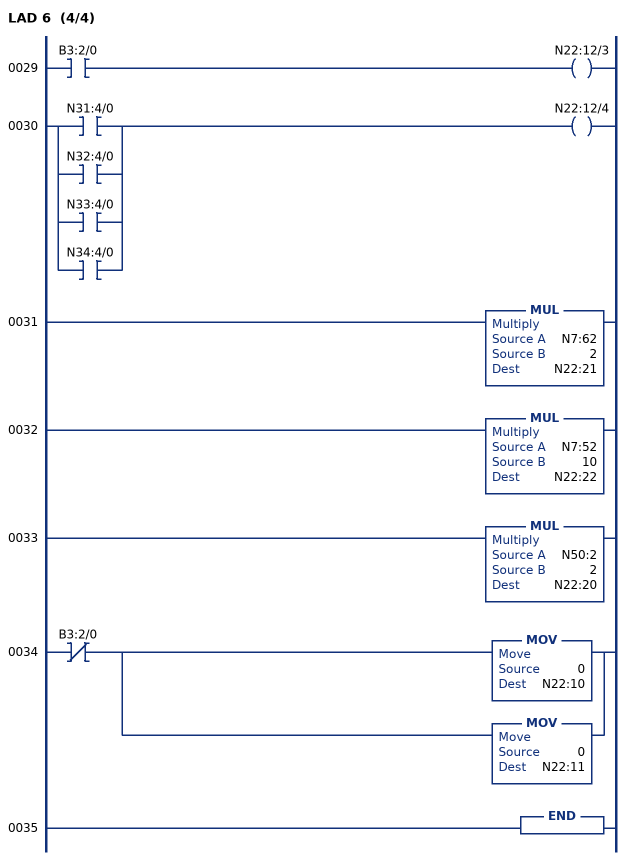
% Rung: 29 %
SOR XIC B3:2/0 OTE N22:12/3 EOR
% Rung: 30 %
SOR BST XIC N31:4/0 NXB XIC N32:4/0 NXB XIC N33:4/0 NXB XIC N34:4/0 BND OTE N22:12/4 EOR
% Rung: 31 %
SOR MUL N7:62 2 N22:21 EOR
% Rung: 32 %
SOR MUL N7:52 10 N22:22 EOR
% Rung: 33 %
SOR MUL N50:2 2 N22:20 EOR
% Rung: 34 %
SOR XIO B3:2/0 BST MOV 0 N22:10 NXB MOV 0 N22:11 BND EOR
% Rung: 35 %
SOR END EOR

LADDER 7
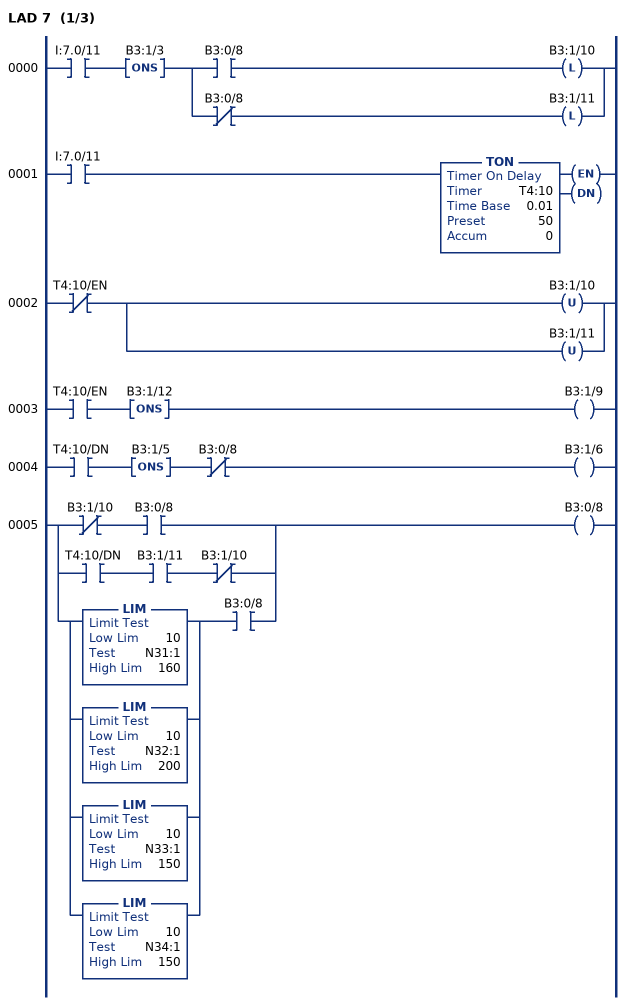
% Rung: 0 %
SOR XIC I:7.0/11 OSR B3:1/3 BST XIC B3:0/8 OTL B3:1/10 NXB XIO B3:0/8 OTL B3:1/11 BND EOR
% Rung: 1 %
SOR XIC I:7.0/11 TON T4:10 0.01 50 0 EOR
% Rung: 2 %
SOR XIO T4:10/EN BST OTU B3:1/10 NXB OTU B3:1/11 BND EOR
% Rung: 3 %
SOR XIC T4:10/EN OSR B3:1/12 OTE B3:1/9 EOR
% Rung: 4 %
SOR XIC T4:10/DN OSR B3:1/5 XIO B3:0/8 OTE B3:1/6 EOR
% Rung: 5 %
SOR BST BST XIO B3:1/10 XIC B3:0/8 NXB XIC T4:10/DN XIC B3:1/11 XIO B3:1/10 BND NXB BST LIM 10 N31:1 160 NXB LIM 10 N32:1 200 NXB LIM 10 N33:1 150 NXB LIM 10 N34:1 150 BND XIC B3:0/8 BND OTE B3:0/8 EOR

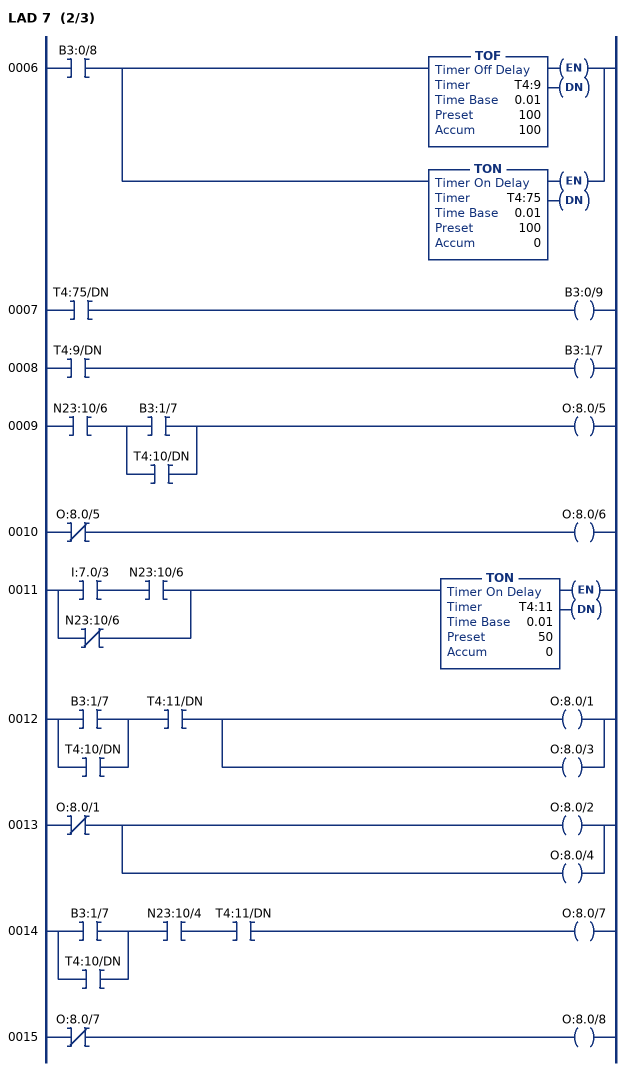
% Rung: 6 %
SOR XIC B3:0/8 BST TOF T4:9 0.01 100 100 NXB TON T4:75 0.01 100 0 BND EOR
% Rung: 7 %
SOR XIC T4:75/DN OTE B3:0/9 EOR
% Rung: 8 %
SOR XIC T4:9/DN OTE B3:1/7 EOR
% Rung: 9 %
SOR XIC N23:10/6 BST XIC B3:1/7 NXB XIC T4:10/DN BND OTE O:8.0/5 EOR
% Rung: 10 %
SOR XIO O:8.0/5 OTE O:8.0/6 EOR
% Rung: 11 %
SOR BST XIC I:7.0/3 XIC N23:10/6 NXB XIO N23:10/6 BND TON T4:11 0.01 50 0 EOR
% Rung: 12 %
SOR BST XIC B3:1/7 NXB XIC T4:10/DN BND XIC T4:11/DN BST OTE O:8.0/1 NXB OTE O:8.0/3 BND EOR
% Rung: 13 %
SOR XIO O:8.0/1 BST OTE O:8.0/2 NXB OTE O:8.0/4 BND EOR
% Rung: 14 %
SOR BST XIC B3:1/7 NXB XIC T4:10/DN BND XIC N23:10/4 XIC T4:11/DN OTE O:8.0/7 EOR
% Rung: 15 %
SOR XIO O:8.0/7 OTE O:8.0/8 EOR

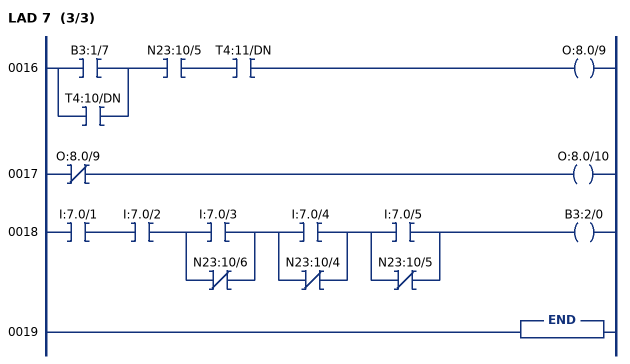
% Rung: 16 %
SOR BST XIC B3:1/7 NXB XIC T4:10/DN BND XIC N23:10/5 XIC T4:11/DN OTE O:8.0/9 EOR
% Rung: 17 %
SOR XIO O:8.0/9 OTE O:8.0/10 EOR
% Rung: 18 %
SOR XIC I:7.0/1 XIC I:7.0/2 BST XIC I:7.0/3 NXB XIO N23:10/6 BND BST XIC I:7.0/4 NXB XIO N23:10/4 BND BST XIC I:7.0/5 NXB XIO N23:10/5 BND OTE B3:2/0 EOR
% Rung: 19 %
SOR END EOR

LADDER 8
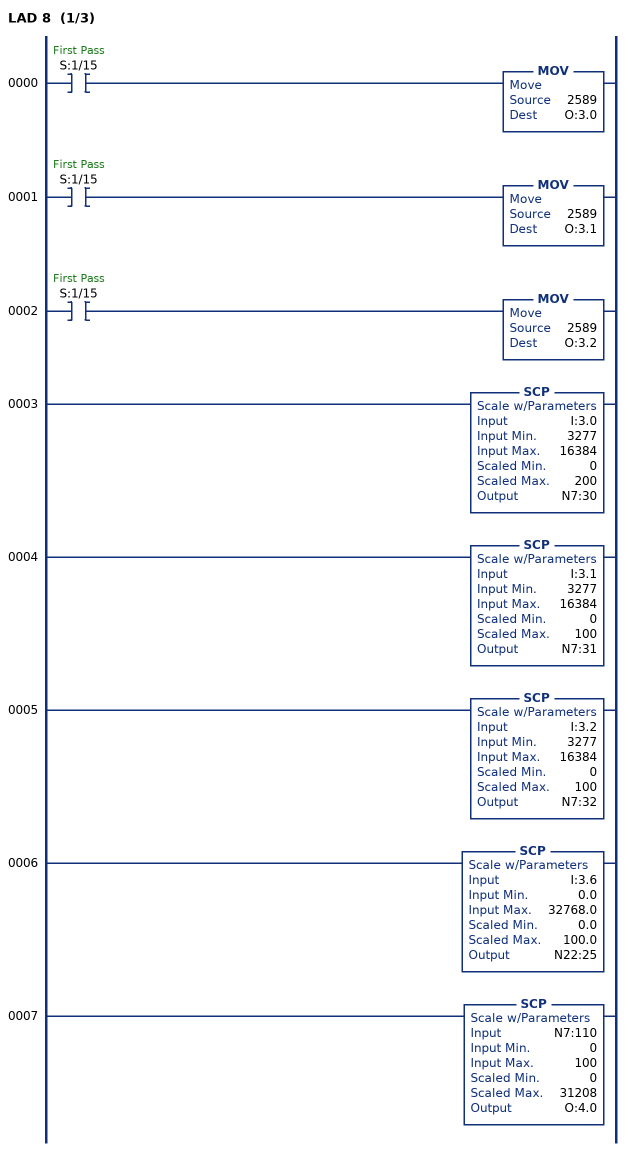
% Rung: 0 %
SOR XIC S:1/15 MOV 2589 O:3.0 EOR
%   S:1/15  "First Pass" %
% Rung: 1 %
SOR XIC S:1/15 MOV 2589 O:3.1 EOR
%   S:1/15  "First Pass" %
% Rung: 2 %
SOR XIC S:1/15 MOV 2589 O:3.2 EOR
%   S:1/15  "First Pass" %
% Rung: 3 %
SOR SCP I:3.0 3277 16384 0 200 N7:30 EOR
% Rung: 4 %
SOR SCP I:3.1 3277 16384 0 100 N7:31 EOR
% Rung: 5 %
SOR SCP I:3.2 3277 16384 0 100 N7:32 EOR
% Rung: 6 %
SOR SCP I:3.6 0.0 32768.0 0.0 100.0 N22:25 EOR
% Rung: 7 %
SOR SCP N7:110 0 100 0 31208 O:4.0 EOR

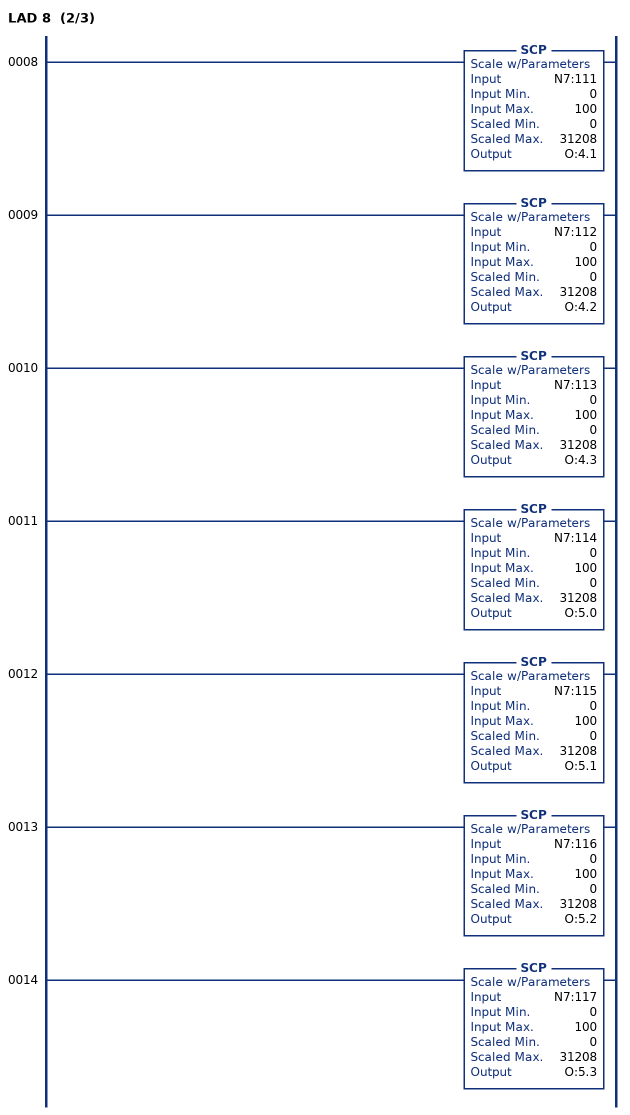
% Rung: 8 %
SOR SCP N7:111 0 100 0 31208 O:4.1 EOR
% Rung: 9 %
SOR SCP N7:112 0 100 0 31208 O:4.2 EOR
% Rung: 10 %
SOR SCP N7:113 0 100 0 31208 O:4.3 EOR
% Rung: 11 %
SOR SCP N7:114 0 100 0 31208 O:5.0 EOR
% Rung: 12 %
SOR SCP N7:115 0 100 0 31208 O:5.1 EOR
% Rung: 13 %
SOR SCP N7:116 0 100 0 31208 O:5.2 EOR
% Rung: 14 %
SOR SCP N7:117 0 100 0 31208 O:5.3 EOR

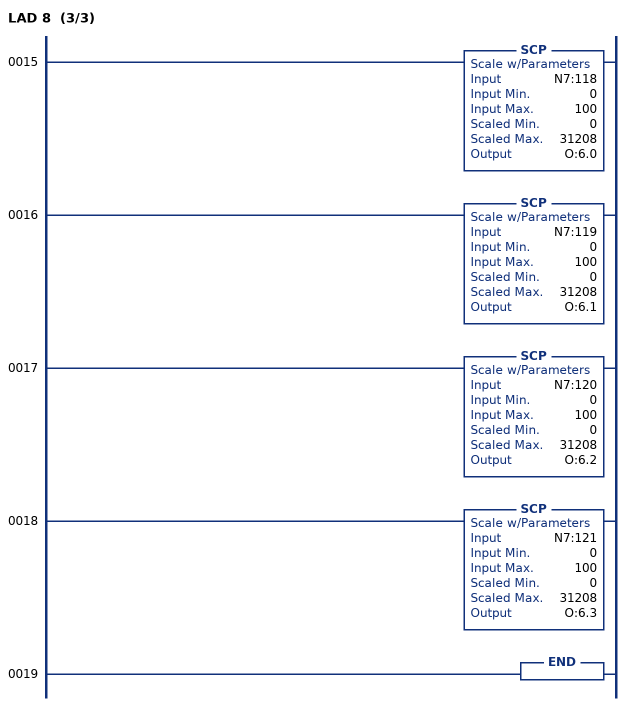
% Rung: 15 %
SOR SCP N7:118 0 100 0 31208 O:6.0 EOR
% Rung: 16 %
SOR SCP N7:119 0 100 0 31208 O:6.1 EOR
% Rung: 17 %
SOR SCP N7:120 0 100 0 31208 O:6.2 EOR
% Rung: 18 %
SOR SCP N7:121 0 100 0 31208 O:6.3 EOR
% Rung: 19 %
SOR END EOR

LADDER 9
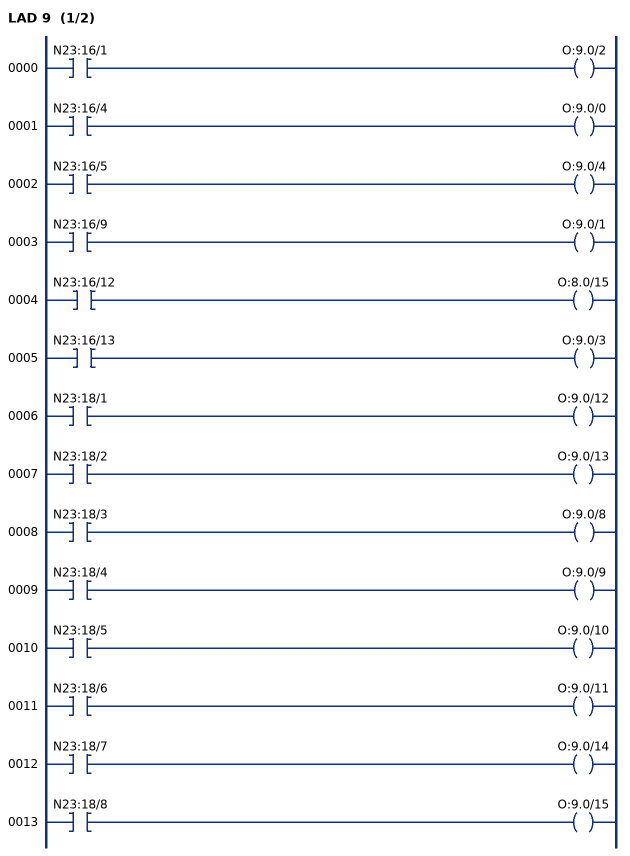
% Rung: 0 %
SOR XIC N23:16/1 OTE O:9.0/2 EOR
% Rung: 1 %
SOR XIC N23:16/4 OTE O:9.0/0 EOR
% Rung: 2 %
SOR XIC N23:16/5 OTE O:9.0/4 EOR
% Rung: 3 %
SOR XIC N23:16/9 OTE O:9.0/1 EOR
% Rung: 4 %
SOR XIC N23:16/12 OTE O:8.0/15 EOR
% Rung: 5 %
SOR XIC N23:16/13 OTE O:9.0/3 EOR
% Rung: 6 %
SOR XIC N23:18/1 OTE O:9.0/12 EOR
% Rung: 7 %
SOR XIC N23:18/2 OTE O:9.0/13 EOR
% Rung: 8 %
SOR XIC N23:18/3 OTE O:9.0/8 EOR
% Rung: 9 %
SOR XIC N23:18/4 OTE O:9.0/9 EOR
% Rung: 10 %
SOR XIC N23:18/5 OTE O:9.0/10 EOR
% Rung: 11 %
SOR XIC N23:18/6 OTE O:9.0/11 EOR
% Rung: 12 %
SOR XIC N23:18/7 OTE O:9.0/14 EOR
% Rung: 13 %
SOR XIC N23:18/8 OTE O:9.0/15 EOR

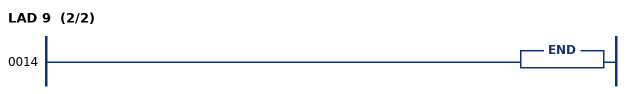
% Rung: 14 %
SOR END EOR

LADDER 10
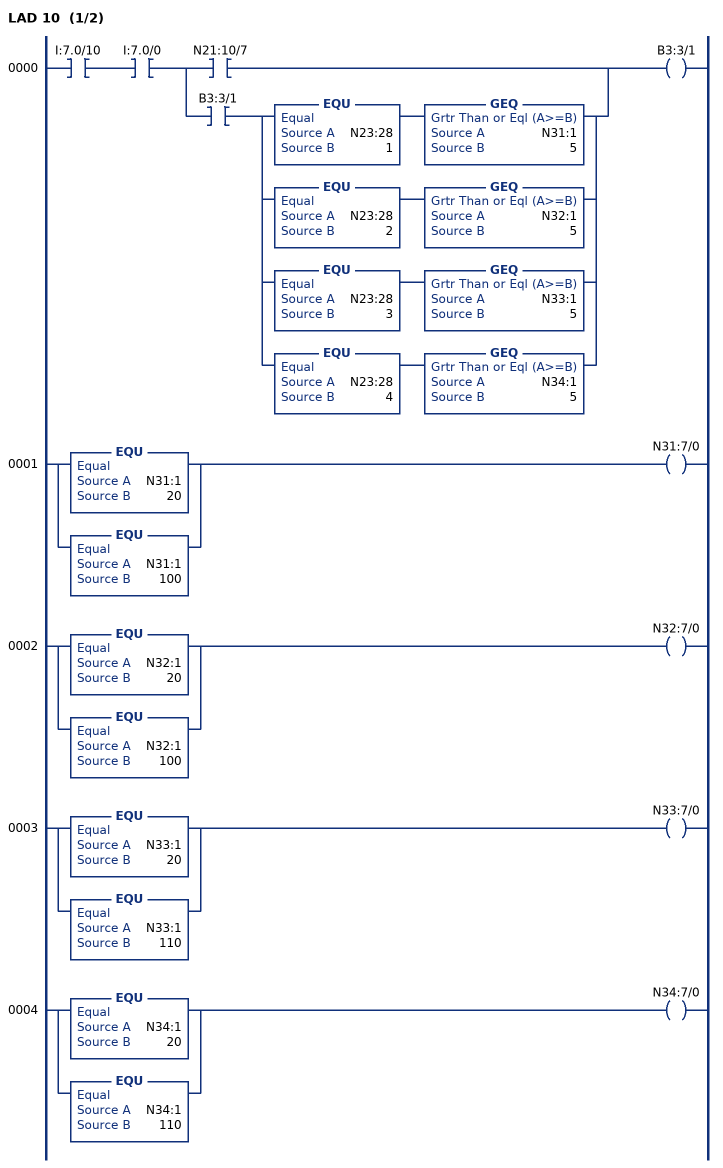
% Rung: 0 %
SOR XIC I:7.0/10 XIC I:7.0/0 BST XIC N21:10/7 NXB XIC B3:3/1 BST EQU N23:28 1 GEQ N31:1 5 NXB EQU N23:28 2 GEQ N32:1 5 NXB EQU N23:28 3 GEQ N33:1 5 NXB EQU N23:28 4 GEQ N34:1 5 BND BND OTE B3:3/1 EOR
% Rung: 1 %
SOR BST EQU N31:1 20 NXB EQU N31:1 100 BND OTE N31:7/0 EOR
% Rung: 2 %
SOR BST EQU N32:1 20 NXB EQU N32:1 100 BND OTE N32:7/0 EOR
% Rung: 3 %
SOR BST EQU N33:1 20 NXB EQU N33:1 110 BND OTE N33:7/0 EOR
% Rung: 4 %
SOR BST EQU N34:1 20 NXB EQU N34:1 110 BND OTE N34:7/0 EOR

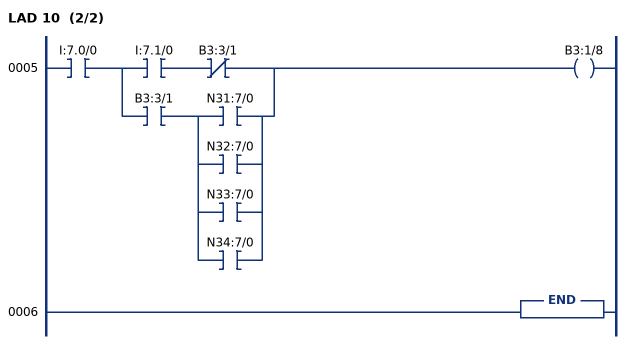
% Rung: 5 %
SOR XIC I:7.0/0 BST XIC I:7.1/0 XIO B3:3/1 NXB XIC B3:3/1 BST XIC N31:7/0 NXB XIC N32:7/0 NXB XIC N33:7/0 NXB XIC N34:7/0 BND BND OTE B3:1/8 EOR
% Rung: 6 %
SOR END EOR

LADDER 11
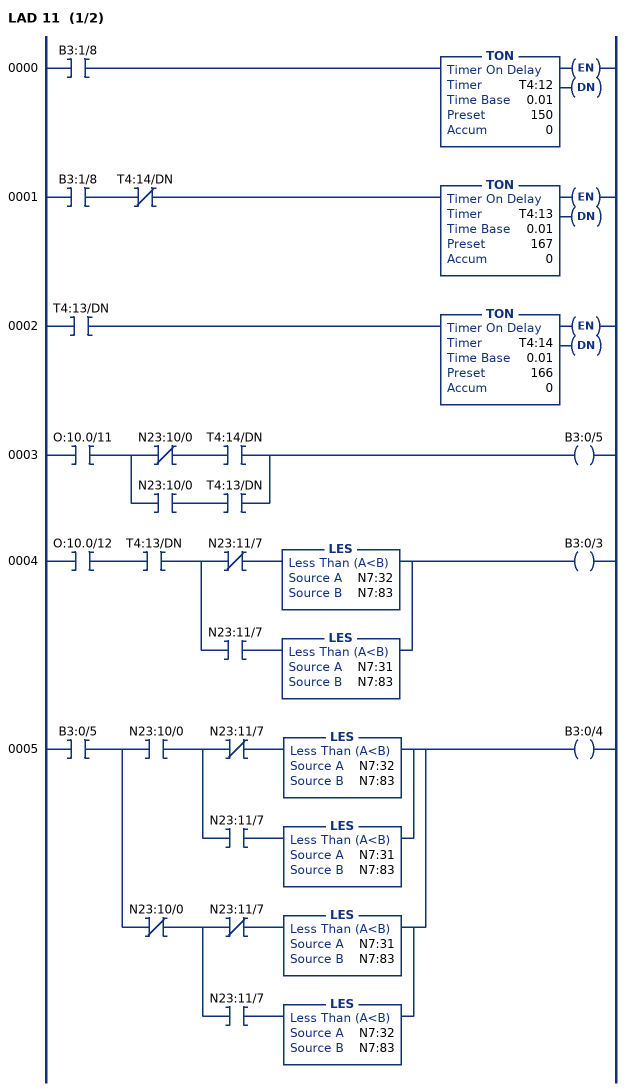
% Rung: 0 %
SOR XIC B3:1/8 TON T4:12 0.01 150 0 EOR
% Rung: 1 %
SOR XIC B3:1/8 XIO T4:14/DN TON T4:13 0.01 167 0 EOR
% Rung: 2 %
SOR XIC T4:13/DN TON T4:14 0.01 166 0 EOR
% Rung: 3 %
SOR XIC O:10.0/11 BST XIO N23:10/0 XIC T4:14/DN NXB XIC N23:10/0 XIC T4:13/DN BND OTE B3:0/5 EOR
% Rung: 4 %
SOR XIC O:10.0/12 XIC T4:13/DN BST XIO N23:11/7 LES N7:32 N7:83 NXB XIC N23:11/7 LES N7:31 N7:83 BND OTE B3:0/3 EOR
% Rung: 5 %
SOR XIC B3:0/5 BST XIC N23:10/0 BST XIO N23:11/7 LES N7:32 N7:83 NXB XIC N23:11/7 LES N7:31 N7:83 BND NXB XIO N23:10/0 BST XIO N23:11/7 LES N7:31 N7:83 NXB XIC N23:11/7 LES N7:32 N7:83 BND BND OTE B3:0/4 EOR

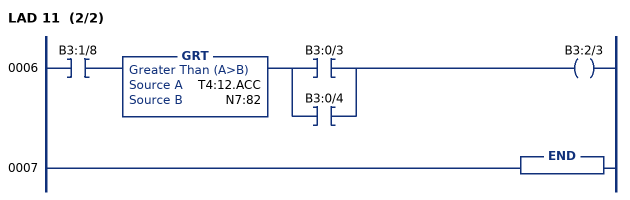
% Rung: 6 %
SOR XIC B3:1/8 GRT T4:12.ACC N7:82 BST XIC B3:0/3 NXB XIC B3:0/4 BND OTE B3:2/3 EOR
% Rung: 7 %
SOR END EOR

LADDER 12
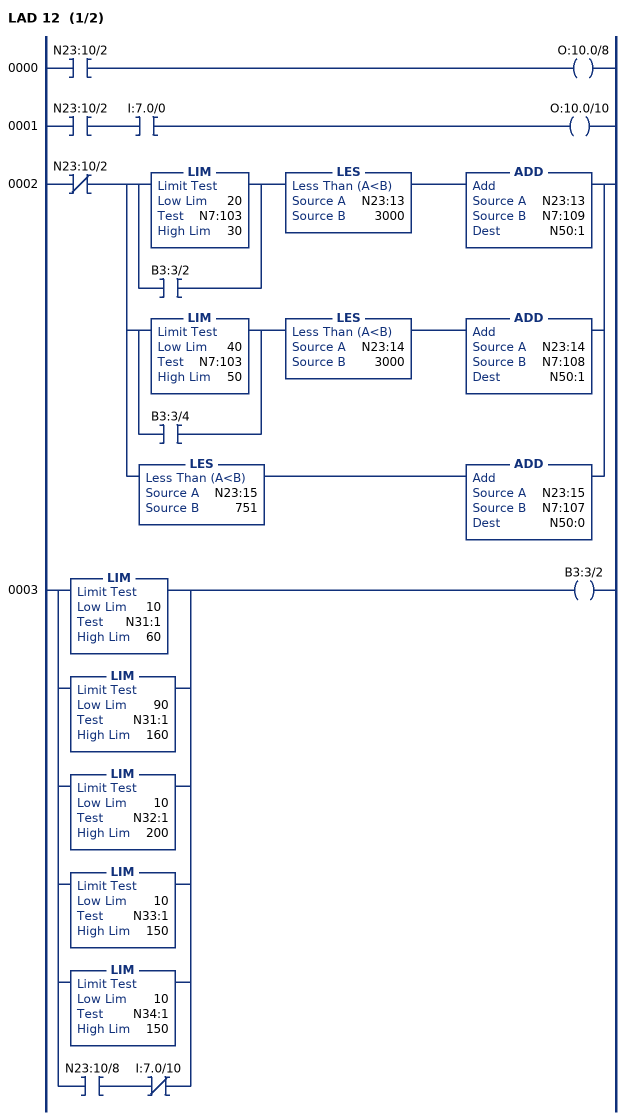
% Rung: 0 %
SOR XIC N23:10/2 OTE O:10.0/8 EOR
% Rung: 1 %
SOR XIC N23:10/2 XIC I:7.0/0 OTE O:10.0/10 EOR
% Rung: 2 %
SOR XIO N23:10/2 BST BST LIM 20 N7:103 30 NXB XIC B3:3/2 BND LES N23:13 3000 ADD N23:13 N7:109 N50:1 NXB BST LIM 40 N7:103 50 NXB XIC B3:3/4 BND LES N23:14 3000 ADD N23:14 N7:108 N50:1 NXB LES N23:15 751 ADD N23:15 N7:107 N50:0 BND EOR
% Rung: 3 %
SOR BST LIM 10 N31:1 60 NXB LIM 90 N31:1 160 NXB LIM 10 N32:1 200 NXB LIM 10 N33:1 150 NXB LIM 10 N34:1 150 NXB XIC N23:10/8 XIO I:7.0/10 BND OTE B3:3/2 EOR

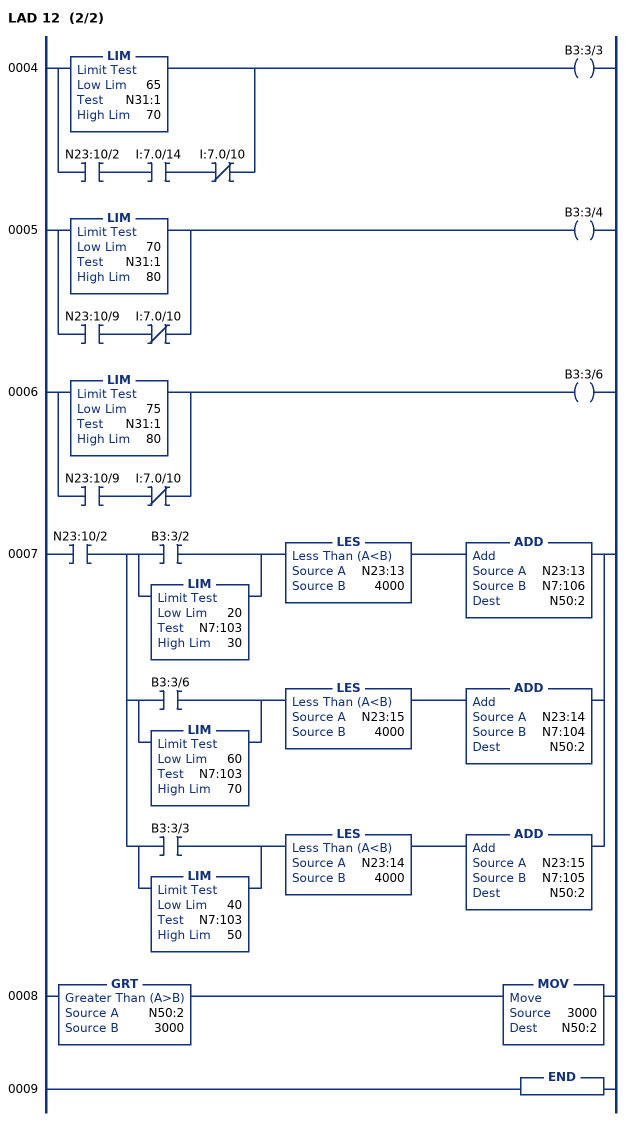
% Rung: 4 %
SOR BST LIM 65 N31:1 70 NXB XIC N23:10/2 XIC I:7.0/14 XIO I:7.0/10 BND OTE B3:3/3 EOR
% Rung: 5 %
SOR BST LIM 70 N31:1 80 NXB XIC N23:10/9 XIO I:7.0/10 BND OTE B3:3/4 EOR
% Rung: 6 %
SOR BST LIM 75 N31:1 80 NXB XIC N23:10/9 XIO I:7.0/10 BND OTE B3:3/6 EOR
% Rung: 7 %
SOR XIC N23:10/2 BST BST XIC B3:3/2 NXB LIM 20 N7:103 30 BND LES N23:13 4000 ADD N23:13 N7:106 N50:2 NXB BST XIC B3:3/6 NXB LIM 60 N7:103 70 BND LES N23:15 4000 ADD N23:14 N7:104 N50:2 NXB BST XIC B3:3/3 NXB LIM 40 N7:103 50 BND LES N23:14 4000 ADD N23:15 N7:105 N50:2 BND EOR
% Rung: 8 %
SOR GRT N50:2 3000 MOV 3000 N50:2 EOR
% Rung: 9 %
SOR END EOR

LADDER 13
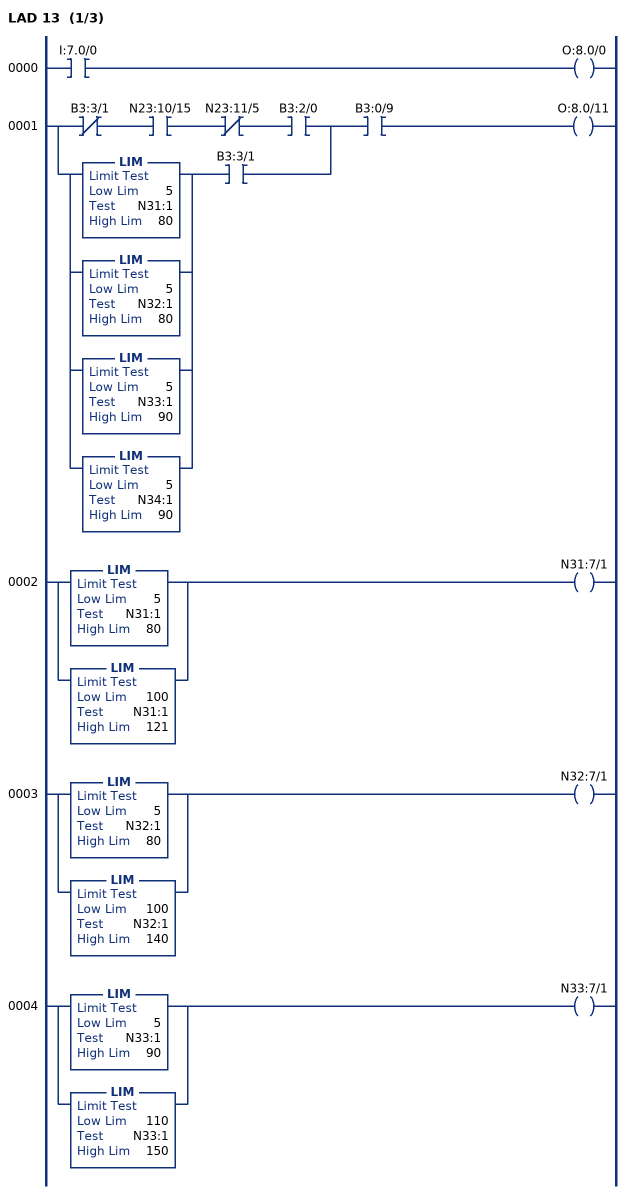
% Rung: 0 %
SOR XIC I:7.0/0 OTE O:8.0/0 EOR
% Rung: 1 %
SOR BST XIO B3:3/1 XIC N23:10/15 XIO N23:11/5 XIC B3:2/0 NXB BST LIM 5 N31:1 80 NXB LIM 5 N32:1 80 NXB LIM 5 N33:1 90 NXB LIM 5 N34:1 90 BND XIC B3:3/1 BND XIC B3:0/9 OTE O:8.0/11 EOR
% Rung: 2 %
SOR BST LIM 5 N31:1 80 NXB LIM 100 N31:1 121 BND OTE N31:7/1 EOR
% Rung: 3 %
SOR BST LIM 5 N32:1 80 NXB LIM 100 N32:1 140 BND OTE N32:7/1 EOR
% Rung: 4 %
SOR BST LIM 5 N33:1 90 NXB LIM 110 N33:1 150 BND OTE N33:7/1 EOR

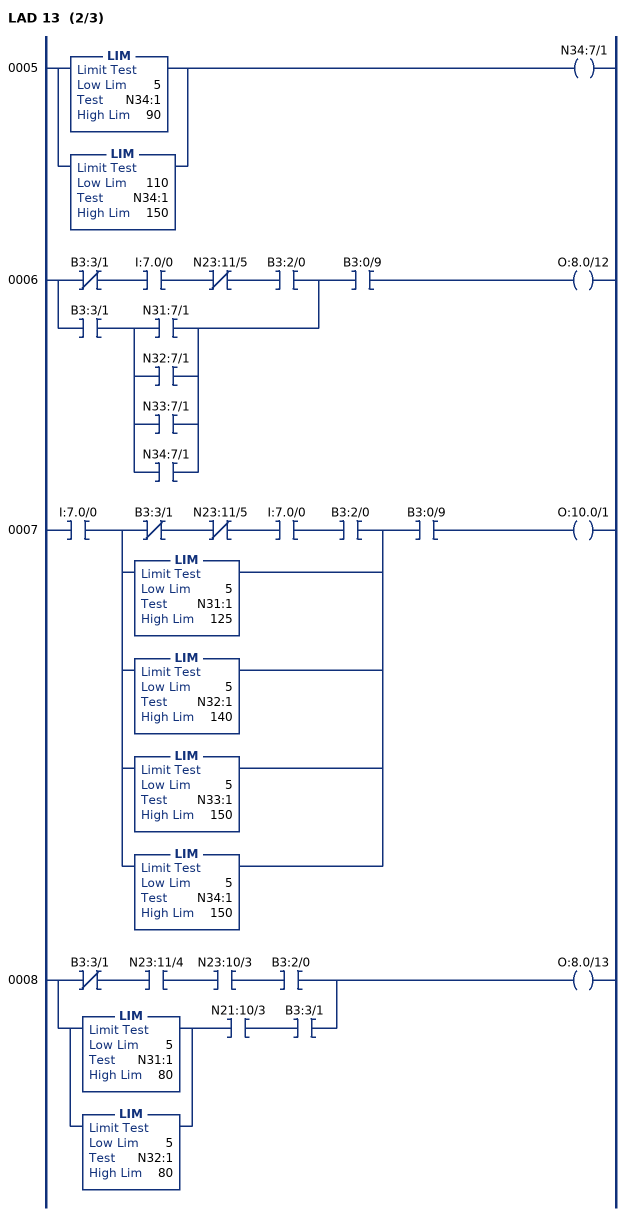
% Rung: 5 %
SOR BST LIM 5 N34:1 90 NXB LIM 110 N34:1 150 BND OTE N34:7/1 EOR
% Rung: 6 %
SOR BST XIO B3:3/1 XIC I:7.0/0 XIO N23:11/5 XIC B3:2/0 NXB XIC B3:3/1 BST XIC N31:7/1 NXB XIC N32:7/1 NXB XIC N33:7/1 NXB XIC N34:7/1 BND BND XIC B3:0/9 OTE O:8.0/12 EOR
% Rung: 7 %
SOR XIC I:7.0/0 BST XIO B3:3/1 XIO N23:11/5 XIC I:7.0/0 XIC B3:2/0 NXB LIM 5 N31:1 125 NXB LIM 5 N32:1 140 NXB LIM 5 N33:1 150 NXB LIM 5 N34:1 150 BND XIC B3:0/9 OTE O:10.0/1 EOR
% Rung: 8 %
SOR BST XIO B3:3/1 XIC N23:11/4 XIC N23:10/3 XIC B3:2/0 NXB BST LIM 5 N31:1 80 NXB LIM 5 N32:1 80 BND XIC N21:10/3 XIC B3:3/1 BND OTE O:8.0/13 EOR

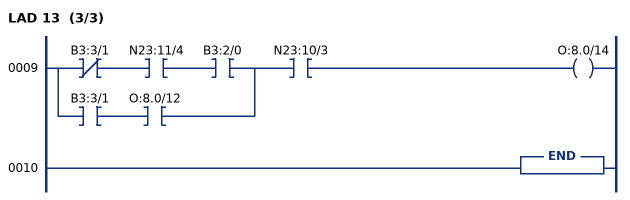
% Rung: 9 %
SOR BST XIO B3:3/1 XIC N23:11/4 XIC B3:2/0 NXB XIC B3:3/1 XIC O:8.0/12 BND XIC N23:10/3 OTE O:8.0/14 EOR
% Rung: 10 %
SOR END EOR

LADDER 14
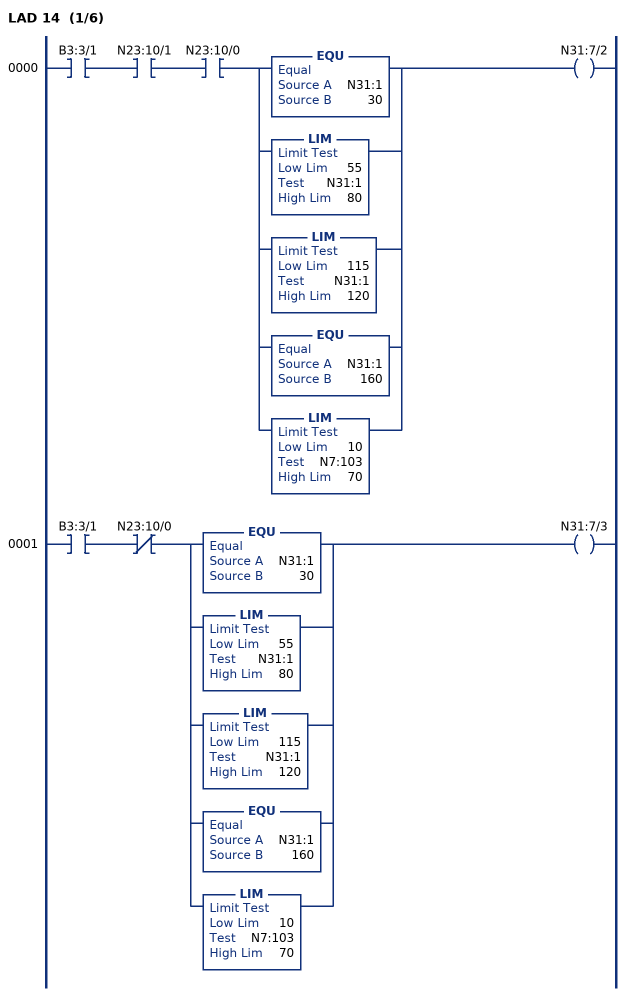
% Rung: 0 %
SOR XIC B3:3/1 XIC N23:10/1 XIC N23:10/0 BST EQU N31:1 30 NXB LIM 55 N31:1 80 NXB LIM 115 N31:1 120 NXB EQU N31:1 160 NXB LIM 10 N7:103 70 BND OTE N31:7/2 EOR
% Rung: 1 %
SOR XIC B3:3/1 XIO N23:10/0 BST EQU N31:1 30 NXB LIM 55 N31:1 80 NXB LIM 115 N31:1 120 NXB EQU N31:1 160 NXB LIM 10 N7:103 70 BND OTE N31:7/3 EOR

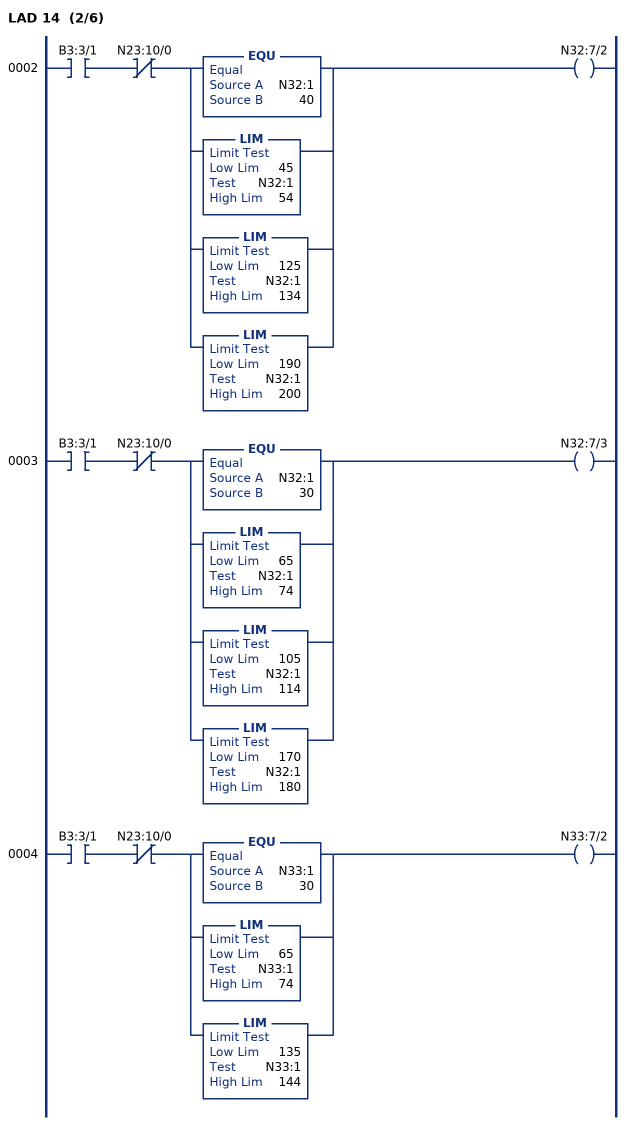
% Rung: 2 %
SOR XIC B3:3/1 XIO N23:10/0 BST EQU N32:1 40 NXB LIM 45 N32:1 54 NXB LIM 125 N32:1 134 NXB LIM 190 N32:1 200 BND OTE N32:7/2 EOR
% Rung: 3 %
SOR XIC B3:3/1 XIO N23:10/0 BST EQU N32:1 30 NXB LIM 65 N32:1 74 NXB LIM 105 N32:1 114 NXB LIM 170 N32:1 180 BND OTE N32:7/3 EOR
% Rung: 4 %
SOR XIC B3:3/1 XIO N23:10/0 BST EQU N33:1 30 NXB LIM 65 N33:1 74 NXB LIM 135 N33:1 144 BND OTE N33:7/2 EOR

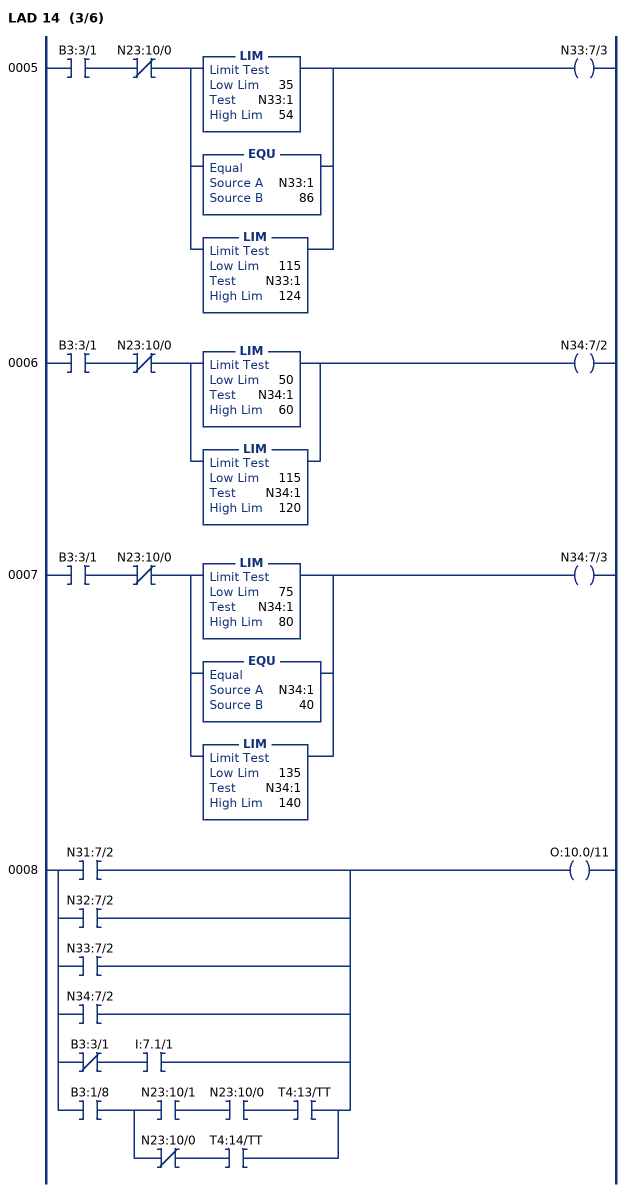
% Rung: 5 %
SOR XIC B3:3/1 XIO N23:10/0 BST LIM 35 N33:1 54 NXB EQU N33:1 86 NXB LIM 115 N33:1 124 BND OTE N33:7/3 EOR
% Rung: 6 %
SOR XIC B3:3/1 XIO N23:10/0 BST LIM 50 N34:1 60 NXB LIM 115 N34:1 120 BND OTE N34:7/2 EOR
% Rung: 7 %
SOR XIC B3:3/1 XIO N23:10/0 BST LIM 75 N34:1 80 NXB EQU N34:1 40 NXB LIM 135 N34:1 140 BND OTE N34:7/3 EOR
% Rung: 8 %
SOR BST XIC N31:7/2 NXB XIC N32:7/2 NXB XIC N33:7/2 NXB XIC N34:7/2 NXB XIO B3:3/1 XIC I:7.1/1 NXB XIC B3:1/8 BST XIC N23:10/1 XIC N23:10/0 XIC T4:13/TT NXB XIO N23:10/0 XIC T4:14/TT BND BND OTE O:10.0/11 EOR

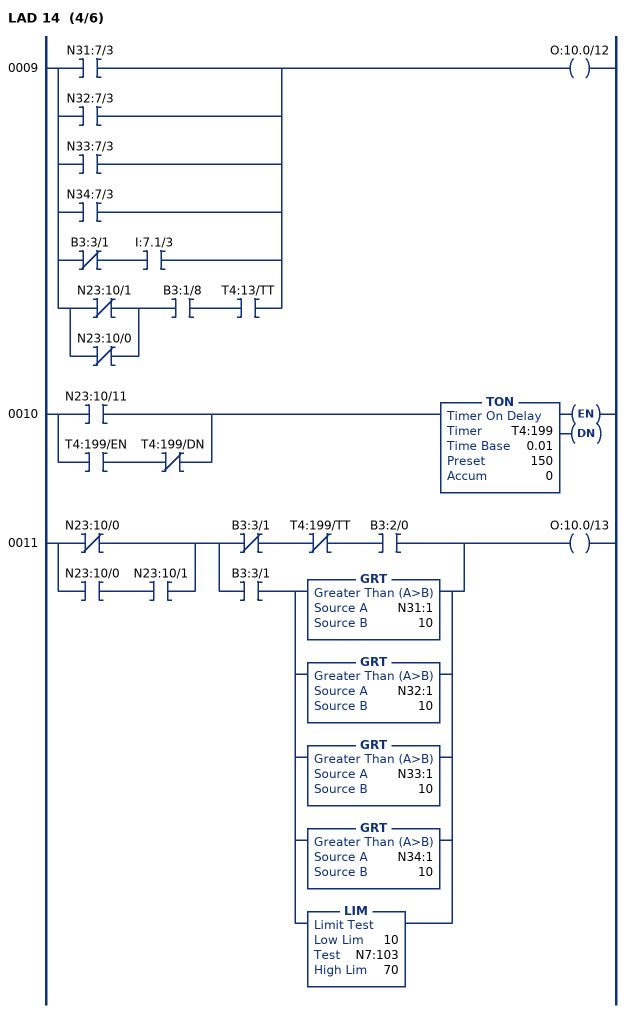
% Rung: 9 %
SOR BST XIC N31:7/3 NXB XIC N32:7/3 NXB XIC N33:7/3 NXB XIC N34:7/3 NXB XIO B3:3/1 XIC I:7.1/3 NXB BST XIO N23:10/1 NXB XIO N23:10/0 BND XIC B3:1/8 XIC T4:13/TT BND OTE O:10.0/12 EOR
% Rung: 10 %
SOR BST XIC N23:10/11 NXB XIC T4:199/EN XIO T4:199/DN BND TON T4:199 0.01 150 0 EOR
% Rung: 11 %
SOR BST XIO N23:10/0 NXB XIC N23:10/0 XIC N23:10/1 BND BST XIO B3:3/1 XIO T4:199/TT XIC B3:2/0 NXB XIC B3:3/1 BST GRT N31:1 10 NXB GRT N32:1 10 NXB GRT N33:1 10 NXB GRT N34:1 10 NXB LIM 10 N7:103 70 BND BND OTE O:10.0/13 EOR

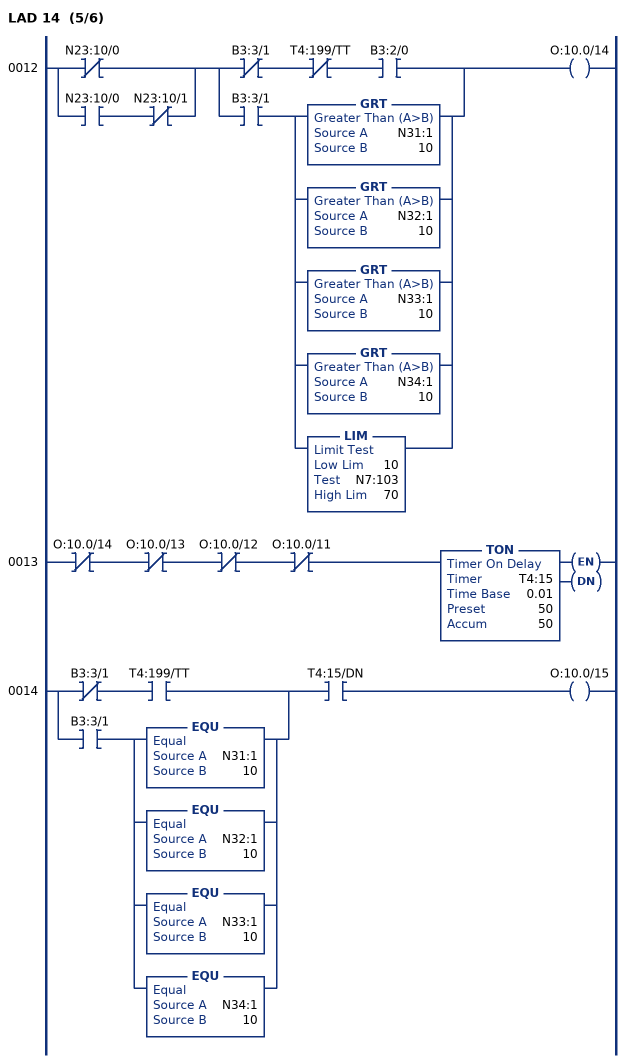
% Rung: 12 %
SOR BST XIO N23:10/0 NXB XIC N23:10/0 XIO N23:10/1 BND BST XIO B3:3/1 XIO T4:199/TT XIC B3:2/0 NXB XIC B3:3/1 BST GRT N31:1 10 NXB GRT N32:1 10 NXB GRT N33:1 10 NXB GRT N34:1 10 NXB LIM 10 N7:103 70 BND BND OTE O:10.0/14 EOR
% Rung: 13 %
SOR XIO O:10.0/14 XIO O:10.0/13 XIO O:10.0/12 XIO O:10.0/11 TON T4:15 0.01 50 50 EOR
% Rung: 14 %
SOR BST XIO B3:3/1 XIC T4:199/TT NXB XIC B3:3/1 BST EQU N31:1 10 NXB EQU N32:1 10 NXB EQU N33:1 10 NXB EQU N34:1 10 BND BND XIC T4:15/DN OTE O:10.0/15 EOR

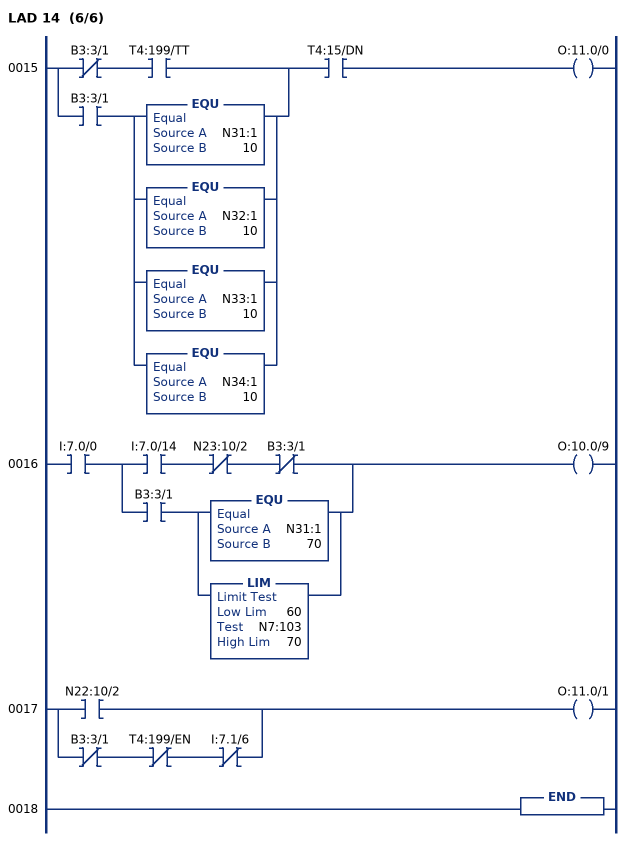
% Rung: 15 %
SOR BST XIO B3:3/1 XIC T4:199/TT NXB XIC B3:3/1 BST EQU N31:1 10 NXB EQU N32:1 10 NXB EQU N33:1 10 NXB EQU N34:1 10 BND BND XIC T4:15/DN OTE O:11.0/0 EOR
% Rung: 16 %
SOR XIC I:7.0/0 BST XIC I:7.0/14 XIO N23:10/2 XIO B3:3/1 NXB XIC B3:3/1 BST EQU N31:1 70 NXB LIM 60 N7:103 70 BND BND OTE O:10.0/9 EOR
% Rung: 17 %
SOR BST XIC N22:10/2 NXB XIO B3:3/1 XIO T4:199/EN XIO I:7.1/6 BND OTE O:11.0/1 EOR
% Rung: 18 %
SOR END EOR

LADDER 15
